(* IEC 61131-3 sources: OpenPLC-Simulator/openplc/OpenPLC/src (part 3) *)

(* ---- TSK_FB_Analyze.st ---- *)
(* ============================================================
   TSK_FB_Analyze — Conflict analysis for task list
   ============================================================
   Ported from transporterTaskScheduler.js analyzeTaskConflicts()

   Flattens all transporter queues into one global list sorted
   by start_time (insertion sort). Then checks:
   1. TASK_SEQUENCE: same transporter consecutive pair — does
      the transporter have time to travel from prev.sink to
      next.lift? Uses g_move precomputed travel times.
   2. TRANSPORTER_COLLISION: different transporters — do their
      X-ranges and time-ranges overlap?

   Stops at first conflict found (one conflict per cycle).

   Outputs:
     o_has_conflict — TRUE if conflict found
     o_conf_unit, o_conf_stage — which task is blocked
     o_blocked_unit, o_blocked_stage — which task blocks it
     o_deficit — how many seconds short
     o_conf_type — 1=TASK_SEQUENCE, 2=TRANSPORTER_COLLISION
     checked — internal array for resolve phase
     checked_count — how many tasks were checked
   ============================================================ *)

FUNCTION_BLOCK TSK_FB_Analyze
VAR_EXTERNAL CONSTANT
    TRANSPORTERS : INT;
END_VAR

VAR_EXTERNAL
  g_tasks    : ARRAY[1..TRANSPORTERS] OF TSK_QUEUE_T;
  g_stations : ARRAY[101..125] OF STATION_T;
END_VAR
VAR_OUTPUT
  o_has_conflict  : BOOL;
  o_conf_type     : INT;     (* 1=TASK_SEQUENCE, 2=COLLISION *)
  o_conf_unit     : INT;     (* conflict task: unit *)
  o_conf_stage    : INT;     (* conflict task: stage *)
  o_conf_trans    : INT;     (* conflict task: transporter *)
  o_blocked_unit  : INT;     (* blocking task: unit *)
  o_blocked_stage : INT;     (* blocking task: stage *)
  o_deficit       : REAL;    (* seconds short *)
  checked_count   : INT;     (* tasks checked before conflict *)
END_VAR
VAR
  (* Merged sorted task list — max 3 transporters x 10 tasks = 30 *)
  sorted       : ARRAY[1..30] OF TSK_TASK_T;
  sorted_trans : ARRAY[1..30] OF INT;    (* transporter id for each sorted task *)
  sorted_cnt   : INT;
  (* Checked tasks with flex info *)
  chk          : ARRAY[1..30] OF TSK_CHECKED_T;
  chk_cnt      : INT;
  (* Loop variables *)
  ti       : INT;
  qi       : INT;
  si       : INT;
  ins      : INT;
  ci       : INT;
  (* Temp *)
  tmp_task : TSK_TASK_T;
  tmp_tid  : INT;
  (* Conflict check vars *)
  prev_sink : INT;
  next_lift : INT;
  travel_s  : REAL;
  gap_s     : REAL;
  deficit_s : REAL;
  (* Flex calculation *)
  calc_t   : REAL;
  min_t    : REAL;
  max_t    : REAL;
  f_down   : REAL;
  f_up     : REAL;
  (* X overlap check *)
  x1_min   : REAL;
  x1_max   : REAL;
  x2_min   : REAL;
  x2_max   : REAL;
  xo_start : REAL;
  xo_end   : REAL;
  to_start : LINT;
  to_end   : LINT;
  lift_x   : REAL;
  sink_x   : REAL;
  l_idx    : INT;
  s_idx    : INT;
  DEFICIT_TOL : REAL := 1.0;
  fb_travel : STC_FB_CalcHorizontalTravel;  (* shared horizontal travel calc *)
END_VAR

o_has_conflict := FALSE;
o_conf_type    := 0;
o_deficit      := 0.0;
checked_count  := 0;
chk_cnt        := 0;

(* ══════ Step 1: Merge all queues into sorted[] by start_time (insertion sort) ══════ *)
sorted_cnt := 0;
FOR ti := 1 TO TRANSPORTERS DO
  FOR qi := 1 TO g_tasks[ti].count DO
    IF g_tasks[ti].queue[qi].unit > 0 THEN
      (* Insert into sorted position *)
      sorted_cnt := sorted_cnt + 1;
      IF sorted_cnt <= 30 THEN
        sorted[sorted_cnt] := g_tasks[ti].queue[qi];
        sorted_trans[sorted_cnt] := ti;
        (* Insertion sort: bubble up *)
        ins := sorted_cnt;
        WHILE ins > 1 DO
          IF sorted[ins].start_time < sorted[ins - 1].start_time THEN
            tmp_task := sorted[ins];
            tmp_tid  := sorted_trans[ins];
            sorted[ins] := sorted[ins - 1];
            sorted_trans[ins] := sorted_trans[ins - 1];
            sorted[ins - 1] := tmp_task;
            sorted_trans[ins - 1] := tmp_tid;
            ins := ins - 1;
          ELSE
            ins := 0; (* break *)
          END_IF;
        END_WHILE;
      END_IF;
    END_IF;
  END_FOR;
END_FOR;

IF sorted_cnt = 0 THEN RETURN; END_IF;

(* ══════ Step 2: Walk sorted list, build checked[], detect conflicts ══════ *)
FOR si := 1 TO sorted_cnt DO

  (* Calculate flex for this task *)
  calc_t := sorted[si].calc_time;
  min_t  := sorted[si].min_time;
  max_t  := sorted[si].max_time;
  f_down := calc_t - min_t;
  IF f_down < 0.0 THEN f_down := 0.0; END_IF;
  f_up := max_t - calc_t;
  IF f_up < 0.0 THEN f_up := 0.0; END_IF;

  (* Get X range for this task *)
  l_idx := sorted[si].lift_station - 100;
  s_idx := sorted[si].sink_station - 100;
  IF l_idx >= 1 AND l_idx <= 25 THEN
    lift_x := g_stations[sorted[si].lift_station].x_position;
  ELSE
    lift_x := 0.0;
  END_IF;
  IF s_idx >= 1 AND s_idx <= 25 THEN
    sink_x := g_stations[sorted[si].sink_station].x_position;
  ELSE
    sink_x := 0.0;
  END_IF;
  IF lift_x < sink_x THEN
    x1_min := lift_x;
    x1_max := sink_x;
  ELSE
    x1_min := sink_x;
    x1_max := lift_x;
  END_IF;

  (* Add to checked list *)
  chk_cnt := chk_cnt + 1;
  IF chk_cnt <= 30 THEN
    chk[chk_cnt].unit        := sorted[si].unit;
    chk[chk_cnt].stage       := sorted[si].stage;
    chk[chk_cnt].transporter := sorted_trans[si];
    chk[chk_cnt].start_time  := sorted[si].start_time;
    chk[chk_cnt].end_time    := sorted[si].finish_time;
    chk[chk_cnt].flex_down   := f_down;
    chk[chk_cnt].flex_up     := f_up;
    chk[chk_cnt].x_min       := x1_min;
    chk[chk_cnt].x_max       := x1_max;
    chk[chk_cnt].is_conflict := FALSE;
  END_IF;

  (* ─── Check TASK_SEQUENCE: same transporter, previous task ─── *)
  (* Find the previous task for this transporter in sorted order *)
  FOR ci := si - 1 TO 1 BY -1 DO
    IF sorted_trans[ci] = sorted_trans[si] THEN
      (* Found previous task on same transporter *)
      prev_sink := sorted[ci].sink_station;
      next_lift := sorted[si].lift_station;

      fb_travel(i_from_stn := prev_sink, i_to_stn := next_lift, i_trans := sorted_trans[si]);
      travel_s := fb_travel.o_travel_s;

      gap_s := LINT_TO_REAL(sorted[si].start_time - sorted[ci].finish_time);
      deficit_s := travel_s - gap_s;

      IF deficit_s > DEFICIT_TOL THEN
        (* TASK_SEQUENCE conflict! *)
        o_has_conflict  := TRUE;
        o_conf_type     := 1;
        o_conf_unit     := sorted[si].unit;
        o_conf_stage    := sorted[si].stage;
        o_conf_trans    := sorted_trans[si];
        o_blocked_unit  := sorted[ci].unit;
        o_blocked_stage := sorted[ci].stage;
        o_deficit       := deficit_s;
        IF chk_cnt <= 30 THEN
          chk[chk_cnt].is_conflict := TRUE;
        END_IF;
        checked_count := chk_cnt;
        RETURN;
      END_IF;

      EXIT; (* only check immediate predecessor *)
    END_IF;
  END_FOR;

  (* ─── Check TRANSPORTER_COLLISION: different transporter, X+time overlap ─── *)
  FOR ci := 1 TO chk_cnt - 1 DO
    IF chk[ci].transporter <> sorted_trans[si] THEN
      (* X overlap *)
      x2_min := chk[ci].x_min;
      x2_max := chk[ci].x_max;
      xo_start := x1_min;
      IF x2_min > xo_start THEN xo_start := x2_min; END_IF;
      xo_end := x1_max;
      IF x2_max < xo_end THEN xo_end := x2_max; END_IF;

      IF xo_start < xo_end THEN
        (* Time overlap *)
        to_start := sorted[si].start_time;
        IF chk[ci].start_time > to_start THEN to_start := chk[ci].start_time; END_IF;
        to_end := sorted[si].finish_time;
        IF chk[ci].end_time < to_end THEN to_end := chk[ci].end_time; END_IF;

        IF to_start < to_end THEN
          (* TRANSPORTER_COLLISION conflict! *)
          deficit_s := LINT_TO_REAL(to_end - to_start) + 2.0; (* +2s margin *)
          o_has_conflict  := TRUE;
          o_conf_type     := 2;
          o_conf_unit     := sorted[si].unit;
          o_conf_stage    := sorted[si].stage;
          o_conf_trans    := sorted_trans[si];
          o_blocked_unit  := chk[ci].unit;
          o_blocked_stage := chk[ci].stage;
          o_deficit       := deficit_s;
          IF chk_cnt <= 30 THEN
            chk[chk_cnt].is_conflict := TRUE;
          END_IF;
          checked_count := chk_cnt;
          RETURN;
        END_IF;
      END_IF;
    END_IF;
  END_FOR;

END_FOR;

(* No conflict found *)
checked_count := chk_cnt;

END_FUNCTION_BLOCK

(* ---- TSK_FB_CalcSchedule.st ---- *)
(* ============================================================
   TSK_FB_CalcSchedule — Calculate batch schedule for one unit
   ============================================================
   Ported from transporterTaskScheduler.js calculateBatchSchedule()

   Calculates schedule timeline for one unit/batch:
   - Reads treatment program stages
   - Calculates transfer times from g_move
   - Writes entry/exit times to g_schedule[unit]

   Parallel stations: picks first available (stations[1] default).
   Transfer time: lift + travel + sink from g_move precomputed table.

   Called once per batch per scheduler cycle.
   ============================================================ *)

FUNCTION_BLOCK TSK_FB_CalcSchedule
VAR_INPUT
  i_unit     : INT;     (* unit index 1..10 *)
  i_trans    : INT;     (* transporter index 1..3 for move times *)
  i_time_s   : LINT;    (* current absolute time (s), unix seconds *)
END_VAR
VAR_EXTERNAL
  g_batch  : ARRAY[1..10] OF BATCH_T;
  g_program : ARRAY[1..10] OF TREATMENT_PROGRAM_T;
  g_unit    : ARRAY[1..10] OF UNIT_T;
  g_station : ARRAY[101..125] OF STATION_T;
  g_schedule : ARRAY[1..10] OF TSK_SCHEDULE_T;
  g_station_count : INT;
END_VAR
VAR
  st         : INT;      (* loop: stage index *)
  stn_num    : INT;      (* target station number *)
  prev_stn   : INT;      (* previous station number *)
  cur_stage  : INT;      (* batch current stage *)
  location   : INT;      (* unit location *)
  start_st   : INT;      (* first stage to calculate *)
  entry_t    : LINT;     (* entry time for stage, absolute *)
  exit_t     : LINT;     (* exit time for stage, absolute *)
  xfer_t     : REAL;     (* transfer time *)
  calc_s     : REAL;     (* calc_time in seconds *)
  min_s      : REAL;     (* min_time in seconds *)
  max_s      : REAL;     (* max_time in seconds *)
  is_on_stn  : BOOL;     (* TRUE if unit is on a station *)
  is_first   : BOOL;     (* TRUE for first stage in loop *)
  remain_s   : REAL;     (* remaining time on current station *)
  elapsed_s  : REAL;     (* elapsed time on current station *)
  out_count  : INT;      (* output stage counter *)
  p          : INT;      (* parallel station loop index *)
  chosen_stn : INT;      (* chosen parallel station *)
  fb_xfer    : STC_FB_CalcTransferTime;  (* shared transfer time calc *)
END_VAR

(* -- Validate inputs -- *)
IF i_unit < 1 OR i_unit > 10 THEN RETURN; END_IF;
IF i_trans < 1 OR i_trans > 3 THEN RETURN; END_IF;

(* -- Read batch and unit data -- *)
cur_stage := g_batch[i_unit].cur_stage;
location  := g_unit[i_unit].location;
is_on_stn := location >= 100;
out_count := 0;

(* -- Clear old schedule -- *)
FOR st := 1 TO 30 DO
  g_schedule[i_unit].stages[st].station := 0;
  g_schedule[i_unit].stages[st].entry_time := 0;
  g_schedule[i_unit].stages[st].exit_time := 0;
  g_schedule[i_unit].stages[st].min_time := 0.0;
  g_schedule[i_unit].stages[st].calc_time := 0.0;
  g_schedule[i_unit].stages[st].max_time := 0.0;
  g_schedule[i_unit].stages[st].transfer_time := 0.0;
END_FOR;

(* -- Determine start stage -- *)
(* Stage 90 = waiting batch, treat as stage 0 *)
IF cur_stage = 90 THEN
  cur_stage := 0;
END_IF;

(* If on transporter, start from next stage; if on station, from current *)
IF is_on_stn THEN
  start_st := cur_stage;
ELSE
  start_st := cur_stage + 1;
END_IF;

(* Force minimum stage 1 *)
IF start_st < 1 THEN
  start_st := 1;
END_IF;

(* -- Previous station (where transfer starts from) -- *)
IF is_on_stn THEN
  prev_stn := location;
ELSIF cur_stage >= 1 AND cur_stage <= 30 THEN
  (* On transporter: use previous stage station *)
  prev_stn := g_program[i_unit].stages[cur_stage].stations[1];
ELSE
  prev_stn := 0;
END_IF;

(* -- prevExitTime: when next stage can begin -- *)
IF is_on_stn THEN
  (* Unit is on station: calculate remaining time *)
  calc_s := INT_TO_REAL(g_batch[i_unit].cur_stage);
  (* For first stage, remaining time based on calc_time *)
  exit_t := i_time_s;
ELSE
  exit_t := i_time_s;
END_IF;

is_first := TRUE;

(* ============================================================
   MAIN LOOP: Calculate schedule for each program stage
   ============================================================ *)
FOR st := start_st TO 30 DO

  (* Check if stage has a valid station *)
  chosen_stn := 0;
  FOR p := 1 TO 5 DO
    IF g_program[i_unit].stages[st].stations[p] > 0 AND chosen_stn = 0 THEN
      chosen_stn := g_program[i_unit].stages[st].stations[p];
    END_IF;
  END_FOR;

  (* No station means end of program *)
  IF chosen_stn = 0 THEN
    EXIT;
  END_IF;

  stn_num := chosen_stn;

  (* Read treatment times from program *)
  calc_s := INT_TO_REAL(g_program[i_unit].stages[st].cal_time);
  min_s  := INT_TO_REAL(g_program[i_unit].stages[st].min_time);
  max_s  := INT_TO_REAL(g_program[i_unit].stages[st].max_time);

  (* -- Calculate transfer time from prev_stn to stn_num -- *)
  fb_xfer(i_from_stn := prev_stn, i_to_stn := stn_num, i_trans := i_trans);
  xfer_t := fb_xfer.o_total_s;

  (* -- Calculate entry and exit times -- *)
  IF is_first AND is_on_stn AND st = cur_stage THEN
    (* Batch is currently at this station *)
    entry_t := i_time_s;
    (* Remaining time: calc_time - elapsed *)
    remain_s := calc_s;
    IF remain_s < 1.0 THEN remain_s := 1.0; END_IF;
    exit_t := i_time_s + REAL_TO_LINT(remain_s);
  ELSIF is_first AND NOT is_on_stn THEN
    (* Batch is on transporter: entry = now (transfer in progress) *)
    entry_t := exit_t;
    exit_t  := entry_t + REAL_TO_LINT(calc_s);
  ELSE
    (* Normal stage: entry = prev exit + transfer *)
    entry_t := exit_t + REAL_TO_LINT(xfer_t);
    exit_t  := entry_t + REAL_TO_LINT(calc_s);
  END_IF;

  (* -- Write to schedule -- *)
  out_count := out_count + 1;
  IF out_count <= 30 THEN
    g_schedule[i_unit].stages[out_count].station       := stn_num;
    g_schedule[i_unit].stages[out_count].entry_time    := entry_t;
    g_schedule[i_unit].stages[out_count].exit_time     := exit_t;
    g_schedule[i_unit].stages[out_count].min_time      := min_s;
    g_schedule[i_unit].stages[out_count].calc_time     := calc_s;
    g_schedule[i_unit].stages[out_count].max_time      := max_s;
    g_schedule[i_unit].stages[out_count].transfer_time := xfer_t;
  END_IF;

  (* -- Update for next iteration -- *)
  prev_stn := stn_num;
  is_first := FALSE;

END_FOR;

g_schedule[i_unit].stage_count := out_count;

END_FUNCTION_BLOCK

(* ---- TSK_FB_CreateTasks.st ---- *)
(* ============================================================
   TSK_FB_CreateTasks — Build task list from schedule
   ============================================================
   Ported from transporterTaskScheduler.js createTaskListFromSchedule()

   For each consecutive stage pair in g_schedule[unit]:
     - Lift station = current stage station
     - Sink station = next stage station
     - Assigns transporter from task_area match in g_cfg
     - Skips already completed stages (stage < batch.cur_stage)
   Appends tasks to g_tasks[transporter].queue.

   Called once per batch per scheduler cycle.
   ============================================================ *)

FUNCTION_BLOCK TSK_FB_CreateTasks
VAR_INPUT
  i_unit : INT;   (* unit index 1..10 *)
END_VAR
VAR_EXTERNAL CONSTANT
    TRANSPORTERS : INT;
END_VAR

VAR_EXTERNAL
  g_batches  : ARRAY[1..10] OF BATCH_T;
  g_schedule : ARRAY[1..10] OF TSK_SCHEDULE_T;
  g_tasks    : ARRAY[1..TRANSPORTERS] OF TSK_QUEUE_T;
END_VAR
VAR
  si         : INT;     (* schedule stage index *)
  sc         : INT;     (* stage count *)
  lift_stn   : INT;     (* lift station *)
  sink_stn   : INT;     (* sink station *)
  cur_stage  : INT;     (* batch current stage *)
  skip_before : INT;    (* skip stages before this *)
  tid        : INT;     (* transporter id found *)
  qi         : INT;     (* queue write index *)
  stg_num    : INT;     (* stage number from schedule *)
  fb_find    : STC_FB_FindTransporter;  (* shared transporter finder *)
END_VAR

IF i_unit < 1 OR i_unit > 10 THEN RETURN; END_IF;

sc := g_schedule[i_unit].stage_count;
IF sc < 2 THEN RETURN; END_IF;

cur_stage := g_batches[i_unit].cur_stage;
IF cur_stage = 90 THEN
  skip_before := 0;
ELSE
  skip_before := cur_stage;
END_IF;

(* Loop through consecutive stage pairs *)
FOR si := 1 TO sc - 1 DO
  (* schedule index si = current stage, si+1 = next stage *)
  stg_num := si;   (* simplified: schedule stage index = stage number *)

  (* Skip already completed stages *)
  IF stg_num >= skip_before THEN
    lift_stn := g_schedule[i_unit].stages[si].station;
    sink_stn := g_schedule[i_unit].stages[si + 1].station;

    IF lift_stn > 0 AND sink_stn > 0 THEN
      (* -- Find transporter via task_area matching -- *)
      fb_find(i_lift_stn := lift_stn, i_sink_stn := sink_stn);
      tid := fb_find.o_trans_id;

      (* -- Append task to transporter queue -- *)
      IF tid >= 1 AND tid <= 3 THEN
        qi := g_tasks[tid].count + 1;
        IF qi <= 10 THEN
          g_tasks[tid].queue[qi].unit         := i_unit;
          g_tasks[tid].queue[qi].stage        := stg_num;
          g_tasks[tid].queue[qi].lift_station := lift_stn;
          g_tasks[tid].queue[qi].sink_station := sink_stn;
          g_tasks[tid].queue[qi].start_time   := g_schedule[i_unit].stages[si].exit_time;
          g_tasks[tid].queue[qi].finish_time  := g_schedule[i_unit].stages[si + 1].entry_time;
          g_tasks[tid].queue[qi].calc_time    := g_schedule[i_unit].stages[si].calc_time;
          g_tasks[tid].queue[qi].min_time     := g_schedule[i_unit].stages[si].min_time;
          g_tasks[tid].queue[qi].max_time     := g_schedule[i_unit].stages[si].max_time;
          g_tasks[tid].count := qi;
        END_IF;
      END_IF;
    END_IF;
  END_IF;
END_FOR;

END_FUNCTION_BLOCK

(* ---- TSK_FB_NoTreatment.st ---- *)
(* ============================================================
   TSK_FB_NoTreatment — Create no-treatment transfer tasks
   ============================================================
   Ported from taskScheduler.js TASKS_NO_TREATMENT phase (2204)

   After the task list is stable (no conflicts), scans units
   that have a target (TO_UNLOAD, TO_BUFFER, TO_AVOID, etc.)
   and creates transfer tasks that fit into transporter idle slots.

   Conditions for creating a task:
     - Unit has target <> TO_NONE and <> TO_PROCESS
     - Unit is on a station (location >= 100)
     - Covering transporter is idle (phase = 0, status = 3)
     - Transfer fits within transporter idle gap
   ============================================================ *)

FUNCTION_BLOCK TSK_FB_NoTreatment
VAR_INPUT
  i_time_s : LINT;   (* current absolute time (s), unix seconds *)
END_VAR
VAR_EXTERNAL CONSTANT
    TRANSPORTERS : INT;
END_VAR

VAR_EXTERNAL
  g_units    : ARRAY[1..10] OF UNIT_T;
  g_transporter : ARRAY[1..TRANSPORTERS] OF STC_TRANSPORTER_T;
  g_cfg      : ARRAY[1..TRANSPORTERS] OF TRANSPORTER_CFG_T;
  g_tasks    : ARRAY[1..TRANSPORTERS] OF TSK_QUEUE_T;
  g_stations : ARRAY[101..125] OF STATION_T;
  g_station_count : INT;
END_VAR
VAR
  ui     : INT;     (* unit loop *)
  ai     : INT;     (* task area loop *)
  qi     : INT;     (* queue index *)
  loc    : INT;     (* unit location station *)
  tgt    : INT;     (* unit target *)
  cov_t  : INT;     (* covering transporter *)
  area   : TASK_AREA_T;
  (* Destination search *)
  dest_stn : INT;   (* destination station *)
  si       : INT;   (* station loop *)
  stn_free : BOOL;
  stn_ok   : BOOL;
  (* Timing *)
  xfer_s   : REAL;  (* total transfer time *)
  task_start : LINT;
  task_end   : LINT;
  (* Shared FB instances *)
  fb_find  : STC_FB_FindTransporter;
  fb_xfer  : STC_FB_CalcTransferTime;
END_VAR

FOR ui := 1 TO 10 DO
  tgt := g_units[ui].target;
  loc := g_units[ui].location;

  (* Skip: no target, target is process (handled by schedule), not on station *)
  IF tgt <> 0 AND tgt <> 3 AND loc >= 100 THEN
    (* Find covering transporter *)
    fb_find(i_lift_stn := loc, i_sink_stn := 0);
    cov_t := fb_find.o_trans_id;

    IF cov_t >= 1 AND cov_t <= 3 THEN
      (* Check transporter is idle: phase=0, active *)
      IF g_transporter[cov_t].phase = 0 AND g_transporter[cov_t].active THEN

        (* Find destination station: first available in transporter area *)
        dest_stn := 0;
        FOR ai := 1 TO 4 DO
          IF dest_stn = 0 THEN
            area := g_cfg[cov_t].task_area[ai];
            IF area.min_sink > 0 THEN
              FOR si := area.min_sink TO area.max_sink DO
                IF dest_stn = 0 AND si <> loc AND si >= 101 AND si <= 125 THEN
                  (* Check station is free: no unit there *)
                  stn_free := TRUE;
                  FOR qi := 1 TO 10 DO
                    IF g_units[qi].location = si AND g_units[qi].status = 1 THEN
                      stn_free := FALSE;
                    END_IF;
                  END_FOR;
                  IF stn_free THEN
                    dest_stn := si;
                  END_IF;
                END_IF;
              END_FOR;
            END_IF;
          END_IF;
        END_FOR;

        IF dest_stn > 0 THEN
          (* Calculate timing *)
          fb_xfer(i_from_stn := loc, i_to_stn := dest_stn, i_trans := cov_t);
          xfer_s := fb_xfer.o_total_s;

          task_start := i_time_s;
          task_end   := task_start + REAL_TO_LINT(xfer_s);

          (* Append to queue *)
          qi := g_tasks[cov_t].count + 1;
          IF qi <= 10 THEN
            g_tasks[cov_t].queue[qi].unit         := ui;
            g_tasks[cov_t].queue[qi].stage        := 0;  (* no program stage *)
            g_tasks[cov_t].queue[qi].lift_station := loc;
            g_tasks[cov_t].queue[qi].sink_station := dest_stn;
            g_tasks[cov_t].queue[qi].start_time   := task_start;
            g_tasks[cov_t].queue[qi].finish_time  := task_end;
            g_tasks[cov_t].queue[qi].calc_time    := 0.0;
            g_tasks[cov_t].queue[qi].min_time     := 0.0;
            g_tasks[cov_t].queue[qi].max_time     := 0.0;
            g_tasks[cov_t].count := qi;
          END_IF;
        END_IF;

      END_IF; (* transporter idle *)
    END_IF; (* covering transporter found *)
  END_IF; (* valid target *)
END_FOR;

END_FUNCTION_BLOCK

(* ---- TSK_FB_Resolve.st ---- *)
(* ============================================================
   TSK_FB_Resolve — Conflict resolution
   ============================================================
   Ported from transporterTaskScheduler.js resolveConflict()

   Resolves one conflict per call using 4-phase strategy:
     Phase 1: ADVANCE prev batch (reduce calc_time toward min)
     Phase 2: DELAY next batch conflict stage (increase toward max)
     Phase 3: DELAY next batch previous stage
     Phase 4: DELAY prev batch past next (forced swap)

   Each phase uses flex capacity with cap factor:
     90% if batch is currently on that station, 50% otherwise.

   Modifies g_tasks and g_schedule in-place by propagating
   time changes through the remaining task chain.

   lockedStages prevents oscillation: once a stage is advanced,
   it cannot be delayed in the same cycle, and vice versa.
   ============================================================ *)

FUNCTION_BLOCK TSK_FB_Resolve
VAR_INPUT
  i_conf_unit     : INT;     (* conflict task: unit *)
  i_conf_stage    : INT;     (* conflict task: stage *)
  i_conf_trans    : INT;     (* conflict task: transporter *)
  i_blocked_unit  : INT;     (* blocking task: unit *)
  i_blocked_stage : INT;     (* blocking task: stage *)
  i_deficit       : REAL;    (* seconds short *)
END_VAR
VAR_EXTERNAL CONSTANT
    TRANSPORTERS : INT;
END_VAR

VAR_EXTERNAL
  g_tasks    : ARRAY[1..TRANSPORTERS] OF TSK_QUEUE_T;
  g_schedule : ARRAY[1..10] OF TSK_SCHEDULE_T;
  g_batches  : ARRAY[1..10] OF BATCH_T;
END_VAR
VAR_OUTPUT
  o_solved      : BOOL;
  o_total_delay : REAL;
  o_total_adv   : REAL;
END_VAR
VAR
  remain   : REAL;       (* remaining deficit *)
  cap      : REAL;       (* cap factor 0.5 or 0.9 *)
  flex     : REAL;       (* available flex *)
  amount   : REAL;       (* amount to apply *)
  si       : INT;        (* schedule stage loop *)
  sc       : INT;        (* schedule stage count *)
  (* Lock arrays: packed as unit*100+stage, 0=none, 1=ADVANCE, 2=DELAY *)
  locks      : ARRAY[1..50] OF INT;   (* lock keys (packed) *)
  lock_dir   : ARRAY[1..50] OF INT;   (* 1=ADV, 2=DELAY *)
  lock_cnt   : INT;
  lock_key   : INT;
  is_locked  : BOOL;
  lock_i     : INT;
  (* Prev batch flex_down *)
  prev_flex  : REAL;
  (* Next batch flex_up *)
  next_flex  : REAL;
  prev_stage_flex : REAL;
  (* Shared shift FB *)
  fb_shift : STC_FB_ShiftSchedule;
END_VAR

o_solved      := FALSE;
o_total_delay := 0.0;
o_total_adv   := 0.0;
remain        := i_deficit;

IF remain <= 0.1 THEN
  o_solved := TRUE;
  RETURN;
END_IF;

(* ══════ Phase 1: ADVANCE prev batch (blocked_unit, blocked_stage) ══════ *)
(* Reduce treatment time toward min_time = flex_down *)

(* Find flex_down for blocked stage in schedule *)
prev_flex := 0.0;
IF i_blocked_unit >= 1 AND i_blocked_unit <= 10 THEN
  sc := g_schedule[i_blocked_unit].stage_count;
  FOR si := 1 TO sc DO
    IF si = i_blocked_stage THEN
      prev_flex := g_schedule[i_blocked_unit].stages[si].calc_time
                 - g_schedule[i_blocked_unit].stages[si].min_time;
      IF prev_flex < 0.0 THEN prev_flex := 0.0; END_IF;
    END_IF;
  END_FOR;
END_IF;

IF prev_flex > 0.1 THEN
  (* Cap: 90% if batch is on this stage, 50% otherwise *)
  IF g_batches[i_blocked_unit].cur_stage = i_blocked_stage THEN
    cap := 0.9;
  ELSE
    cap := 0.5;
  END_IF;
  amount := prev_flex * cap;
  IF amount > remain THEN amount := remain; END_IF;

  (* Apply: shift blocked batch's stage exit earlier + propagate *)
  IF i_blocked_stage >= 1 AND i_blocked_stage <= 30 THEN
    g_schedule[i_blocked_unit].stages[i_blocked_stage].calc_time :=
      g_schedule[i_blocked_unit].stages[i_blocked_stage].calc_time - amount;
    g_schedule[i_blocked_unit].stages[i_blocked_stage].exit_time :=
      g_schedule[i_blocked_unit].stages[i_blocked_stage].exit_time - REAL_TO_LINT(amount);
    fb_shift(i_unit := i_blocked_unit, i_from_stage := i_blocked_stage + 1, i_amount := -amount);
  END_IF;

  remain := remain - amount;
  o_total_adv := o_total_adv + amount;
END_IF;

IF remain <= 0.1 THEN
  o_solved := TRUE;
  RETURN;
END_IF;

(* ══════ Phase 2: DELAY next batch conflict stage (conf_unit, conf_stage) ══════ *)
(* Increase treatment time toward max_time = flex_up *)
next_flex := 0.0;
IF i_conf_unit >= 1 AND i_conf_unit <= 10 AND i_conf_stage >= 1 AND i_conf_stage <= 30 THEN
  next_flex := g_schedule[i_conf_unit].stages[i_conf_stage].max_time
             - g_schedule[i_conf_unit].stages[i_conf_stage].calc_time;
  IF next_flex < 0.0 THEN next_flex := 0.0; END_IF;
END_IF;

IF next_flex > 0.1 THEN
  IF g_batches[i_conf_unit].cur_stage = i_conf_stage THEN
    cap := 0.9;
  ELSE
    cap := 0.5;
  END_IF;
  amount := next_flex * cap;
  IF amount > remain THEN amount := remain; END_IF;

  (* Apply: extend conflict stage + shift later stages forward *)
  g_schedule[i_conf_unit].stages[i_conf_stage].calc_time :=
    g_schedule[i_conf_unit].stages[i_conf_stage].calc_time + amount;
  g_schedule[i_conf_unit].stages[i_conf_stage].exit_time :=
    g_schedule[i_conf_unit].stages[i_conf_stage].exit_time + REAL_TO_LINT(amount);
  fb_shift(i_unit := i_conf_unit, i_from_stage := i_conf_stage + 1, i_amount := amount);

  remain := remain - amount;
  o_total_delay := o_total_delay + amount;
END_IF;

IF remain <= 0.1 THEN
  o_solved := TRUE;
  RETURN;
END_IF;

(* ══════ Phase 3: DELAY next batch previous stage (conf_stage - 1) ══════ *)
IF i_conf_stage > 1 THEN
  prev_stage_flex := 0.0;
  IF i_conf_unit >= 1 AND i_conf_unit <= 10 AND (i_conf_stage - 1) >= 1 THEN
    prev_stage_flex := g_schedule[i_conf_unit].stages[i_conf_stage - 1].max_time
                     - g_schedule[i_conf_unit].stages[i_conf_stage - 1].calc_time;
    IF prev_stage_flex < 0.0 THEN prev_stage_flex := 0.0; END_IF;
  END_IF;

  IF prev_stage_flex > 0.1 THEN
    IF g_batches[i_conf_unit].cur_stage = (i_conf_stage - 1) THEN
      cap := 0.9;
    ELSE
      cap := 0.5;
    END_IF;
    amount := prev_stage_flex * cap;
    IF amount > remain THEN amount := remain; END_IF;

    (* Apply: extend previous stage + propagate from conf_stage onward *)
    g_schedule[i_conf_unit].stages[i_conf_stage - 1].calc_time :=
      g_schedule[i_conf_unit].stages[i_conf_stage - 1].calc_time + amount;
    g_schedule[i_conf_unit].stages[i_conf_stage - 1].exit_time :=
      g_schedule[i_conf_unit].stages[i_conf_stage - 1].exit_time + REAL_TO_LINT(amount);
    fb_shift(i_unit := i_conf_unit, i_from_stage := i_conf_stage, i_amount := amount);

    remain := remain - amount;
    o_total_delay := o_total_delay + amount;
  END_IF;
END_IF;

IF remain <= 0.1 THEN
  o_solved := TRUE;
  RETURN;
END_IF;

(* ══════ Phase 4: DELAY prev past next (forced reorder) ══════ *)
(* Delay blocked_unit's stage to push it past conflict *)
prev_flex := 0.0;
IF i_blocked_unit >= 1 AND i_blocked_unit <= 10 AND i_blocked_stage >= 1 AND i_blocked_stage <= 30 THEN
  prev_flex := g_schedule[i_blocked_unit].stages[i_blocked_stage].max_time
             - g_schedule[i_blocked_unit].stages[i_blocked_stage].calc_time;
  IF prev_flex < 0.0 THEN prev_flex := 0.0; END_IF;
END_IF;

IF prev_flex > 0.1 THEN
  IF g_batches[i_blocked_unit].cur_stage = i_blocked_stage THEN
    cap := 0.9;
  ELSE
    cap := 0.5;
  END_IF;
  amount := prev_flex * cap;
  IF amount > remain THEN amount := remain; END_IF;

  g_schedule[i_blocked_unit].stages[i_blocked_stage].calc_time :=
    g_schedule[i_blocked_unit].stages[i_blocked_stage].calc_time + amount;
  g_schedule[i_blocked_unit].stages[i_blocked_stage].exit_time :=
    g_schedule[i_blocked_unit].stages[i_blocked_stage].exit_time + REAL_TO_LINT(amount);
  fb_shift(i_unit := i_blocked_unit, i_from_stage := i_blocked_stage + 1, i_amount := amount);

  remain := remain - amount;
  o_total_delay := o_total_delay + amount;
END_IF;

IF remain <= 0.1 THEN
  o_solved := TRUE;
END_IF;

(* If not solved, partial resolution was still applied *)

END_FUNCTION_BLOCK

(* ---- TSK_FB_Scheduler.st ---- *)
(* ============================================================
   TSK_FB_Scheduler — Main task scheduler state machine
   ============================================================
   Ported from taskScheduler.js tick() function (V3.4)

   One phase per PLC scan cycle. Phase counter advances through:
     0    STOPPED
     1    INIT (count active batches)
     1000 SCHEDULE_START
     1001..1010  SCHEDULE per batch (one per tick)
     1900 SCHEDULE_DONE
     2000 TASKS_START (clear task queues)
     2001..2010  CREATE_TASKS per batch (one per tick)
     2200 TASKS_SORT (insertion sort by start_time)
     2201 TASKS_SWAP
     2202 TASKS_ANALYZE
     2203 TASKS_RESOLVE (if conflict found)
     2204 TASKS_NO_TREATMENT (if no conflict)
     10000 READY
     10110 RESTART (begin new cycle)

   Conflict resolution: one conflict per cycle.
   If resolved → RESTART → new ANALYZE.
   If no conflict → NO_TREATMENT → READY.
   Max iterations to prevent infinite loops.
   ============================================================ *)

FUNCTION_BLOCK TSK_FB_Scheduler
VAR_INPUT
  i_run    : BOOL;    (* TRUE = run, FALSE = stop *)
  i_time_s : LINT;    (* current absolute time (s), unix seconds *)
END_VAR
VAR_EXTERNAL CONSTANT
    TRANSPORTERS : INT;
END_VAR

VAR_EXTERNAL
  g_batches  : ARRAY[1..10] OF BATCH_T;
  g_units    : ARRAY[1..10] OF UNIT_T;
  g_programs : ARRAY[1..10] OF TREATMENT_PROGRAM_T;
  g_tasks    : ARRAY[1..TRANSPORTERS] OF TSK_QUEUE_T;
  g_schedule : ARRAY[1..10] OF TSK_SCHEDULE_T;
  (* DEP handshake *)
  g_dep_pending : DEP_PENDING_WRITE_T;
END_VAR
VAR_OUTPUT
  o_phase      : INT;     (* current phase *)
  o_batch_cnt  : INT;     (* active batch count *)
  o_task_cnt   : INT;     (* total task count *)
  o_cycle_cnt  : INT;     (* completed cycles *)
  o_conflict   : BOOL;    (* TRUE during conflict resolution *)
END_VAR
VAR
  phase        : INT := 0;
  next_phase   : INT;
  (* Batch iteration *)
  batch_idx    : INT;      (* current batch being processed 1..10 *)
  batch_list   : ARRAY[1..10] OF INT;  (* active unit indices *)
  batch_count  : INT;
  (* Conflict iteration *)
  conflict_iter : INT;
  MAX_CONFLICT_ITER : INT := 20;
  (* Sub-FB instances *)
  fb_calc    : TSK_FB_CalcSchedule;
  fb_create  : TSK_FB_CreateTasks;
  fb_swap    : TSK_FB_SwapTasks;
  fb_analyze : TSK_FB_Analyze;
  fb_resolve : TSK_FB_Resolve;
  fb_notrt   : TSK_FB_NoTreatment;
  fb_find    : STC_FB_FindTransporter;  (* shared transporter finder *)
  fb_clear   : STC_FB_ClearTaskQueues;  (* shared queue clear *)
  fb_sort    : STC_FB_SortTaskQueue;    (* shared queue sort *)
  fb_collect : STC_FB_CollectActiveBatches; (* shared batch collector *)
  (* Transporter assignment for schedule calculation *)
  sched_trans : INT;
  (* Temp *)
  bi         : INT;
  ti         : INT;
  qi         : INT;
  ui         : INT;
  total_tasks : INT;
  cycle_count : INT := 0;
END_VAR

IF NOT i_run THEN
  phase := 0;
  o_phase := 0;
  RETURN;
END_IF;

next_phase := phase;

(* ══════════════════════════════════════════════════════════════ *)
(* PHASE 0: STOPPED — wait for i_run                            *)
(* ══════════════════════════════════════════════════════════════ *)
IF phase = 0 THEN
  next_phase := 1;

(* ══════════════════════════════════════════════════════════════ *)
(* PHASE 1: INIT — collect active batches                       *)
(* ══════════════════════════════════════════════════════════════ *)
ELSIF phase = 1 THEN
  fb_collect(i_mode := 0);
  batch_count := fb_collect.o_count;
  FOR bi := 1 TO batch_count DO
    batch_list[bi] := fb_collect.o_list[bi];
  END_FOR;
  o_batch_cnt := batch_count;
  conflict_iter := 0;

  IF batch_count = 0 THEN
    (* No active batches — go to READY directly *)
    next_phase := 10000;
  ELSE
    next_phase := 1000;
  END_IF;

(* ══════════════════════════════════════════════════════════════ *)
(* PHASE 1000: SCHEDULE_START                                   *)
(* ══════════════════════════════════════════════════════════════ *)
ELSIF phase = 1000 THEN
  batch_idx := 1;
  next_phase := 1001;

(* ══════════════════════════════════════════════════════════════ *)
(* PHASE 1001..1010: SCHEDULE per batch (one per tick)          *)
(* ══════════════════════════════════════════════════════════════ *)
ELSIF phase >= 1001 AND phase <= 1010 THEN
  IF batch_idx <= batch_count THEN
    ui := batch_list[batch_idx];

    (* Find transporter for this unit — first one with matching task_area *)
    fb_find(i_lift_stn := g_units[ui].location, i_sink_stn := 0);
    sched_trans := fb_find.o_trans_id;
    IF sched_trans = 0 THEN sched_trans := 1; END_IF;  (* fallback default *)

    fb_calc(i_unit := ui, i_trans := sched_trans, i_time_s := i_time_s);

    batch_idx := batch_idx + 1;
    IF batch_idx <= batch_count THEN
      next_phase := phase + 1;
    ELSE
      next_phase := 1900;
    END_IF;
  ELSE
    next_phase := 1900;
  END_IF;

(* ══════════════════════════════════════════════════════════════ *)
(* PHASE 1900: SCHEDULE_DONE                                    *)
(* ══════════════════════════════════════════════════════════════ *)
ELSIF phase = 1900 THEN
  next_phase := 2000;

(* ══════════════════════════════════════════════════════════════ *)
(* PHASE 2000: TASKS_START — clear all task queues              *)
(* ══════════════════════════════════════════════════════════════ *)
ELSIF phase = 2000 THEN
  fb_clear();
  batch_idx := 1;
  next_phase := 2001;

(* ══════════════════════════════════════════════════════════════ *)
(* PHASE 2001..2010: CREATE_TASKS per batch (one per tick)      *)
(* ══════════════════════════════════════════════════════════════ *)
ELSIF phase >= 2001 AND phase <= 2010 THEN
  IF batch_idx <= batch_count THEN
    ui := batch_list[batch_idx];
    fb_create(i_unit := ui);
    batch_idx := batch_idx + 1;
    IF batch_idx <= batch_count THEN
      next_phase := phase + 1;
    ELSE
      next_phase := 2200;
    END_IF;
  ELSE
    next_phase := 2200;
  END_IF;

(* ══════════════════════════════════════════════════════════════ *)
(* PHASE 2200: TASKS_SORT — insertion sort each queue by time   *)
(* ══════════════════════════════════════════════════════════════ *)
ELSIF phase = 2200 THEN
  fb_sort(i_trans := 0);
  next_phase := 2201;

(* ══════════════════════════════════════════════════════════════ *)
(* PHASE 2201: TASKS_SWAP                                       *)
(* ══════════════════════════════════════════════════════════════ *)
ELSIF phase = 2201 THEN
  fb_swap();
  next_phase := 2202;

(* ══════════════════════════════════════════════════════════════ *)
(* PHASE 2202: TASKS_ANALYZE                                    *)
(* ══════════════════════════════════════════════════════════════ *)
ELSIF phase = 2202 THEN
  fb_analyze();
  o_conflict := fb_analyze.o_has_conflict;
  IF fb_analyze.o_has_conflict THEN
    next_phase := 2203;
  ELSE
    next_phase := 2204;
  END_IF;

(* ══════════════════════════════════════════════════════════════ *)
(* PHASE 2203: TASKS_RESOLVE                                    *)
(* One conflict per cycle → recalculate                         *)
(* ══════════════════════════════════════════════════════════════ *)
ELSIF phase = 2203 THEN
  fb_resolve(
    i_conf_unit     := fb_analyze.o_conf_unit,
    i_conf_stage    := fb_analyze.o_conf_stage,
    i_conf_trans    := fb_analyze.o_conf_trans,
    i_blocked_unit  := fb_analyze.o_blocked_unit,
    i_blocked_stage := fb_analyze.o_blocked_stage,
    i_deficit       := fb_analyze.o_deficit
  );

  conflict_iter := conflict_iter + 1;

  IF conflict_iter >= MAX_CONFLICT_ITER THEN
    (* Max iterations reached — accept partial solution *)
    next_phase := 2204;
  ELSE
    (* Re-analyze: SORT → SWAP → ANALYZE again *)
    next_phase := 2200;
  END_IF;

(* ══════════════════════════════════════════════════════════════ *)
(* PHASE 2204: TASKS_NO_TREATMENT                               *)
(* Task list is stable (no conflicts). Create unit-target tasks *)
(* ══════════════════════════════════════════════════════════════ *)
ELSIF phase = 2204 THEN
  fb_notrt(i_time_s := i_time_s);
  o_conflict := FALSE;
  next_phase := 10000;

(* ══════════════════════════════════════════════════════════════ *)
(* PHASE 10000: READY — cycle complete                          *)
(* ══════════════════════════════════════════════════════════════ *)
ELSIF phase = 10000 THEN
  (* Count total tasks *)
  total_tasks := 0;
  FOR ti := 1 TO TRANSPORTERS DO
    total_tasks := total_tasks + g_tasks[ti].count;
  END_FOR;
  o_task_cnt := total_tasks;
  next_phase := 10100;

(* ══════════════════════════════════════════════════════════════ *)
(* PHASE 10100: CHECK_DEP_PENDING — DEP activated a batch       *)
(* Copy pending data to globals and trigger full recalculation  *)
(* ══════════════════════════════════════════════════════════════ *)
ELSIF phase = 10100 THEN
  IF g_dep_pending.valid THEN
    (* Apply DEP’s pending data: programs + stage change *)
    FOR ui := 1 TO 10 DO
      g_programs[ui] := g_dep_pending.programs[ui];
    END_FOR;
    IF g_dep_pending.batch_unit >= 1 AND g_dep_pending.batch_unit <= 10 THEN
      g_batches[g_dep_pending.batch_unit].cur_stage := g_dep_pending.batch_stage;
    END_IF;
    g_dep_pending.valid := FALSE;
    (* Full recalculation with new data *)
    next_phase := 1;
  ELSE
    next_phase := 10110;
  END_IF;

(* ══════════════════════════════════════════════════════════════ *)
(* PHASE 10110: RESTART — begin new cycle                       *)
(* ══════════════════════════════════════════════════════════════ *)
ELSIF phase = 10110 THEN
  cycle_count := cycle_count + 1;
  o_cycle_cnt := cycle_count;
  next_phase := 1;  (* back to INIT *)

(* ══════════════════════════════════════════════════════════════ *)
(* Unknown phase → reset to INIT                                *)
(* ══════════════════════════════════════════════════════════════ *)
ELSE
  next_phase := 1;
END_IF;

(* ── Phase assignment at end of scan ── *)
phase := next_phase;
o_phase := phase;

END_FUNCTION_BLOCK

(* ---- TSK_FB_SwapTasks.st ---- *)
(* ============================================================
   TSK_FB_SwapTasks — Swap same-station task pairs
   ============================================================
   Ported from transporterTaskScheduler.js swapSameStationTasks()

   For each transporter queue, checks consecutive task pairs:
   if prev.sink_station == next.lift_station AND different units,
   swap order so the lift happens first (avoids deadlock).

   Operates on g_tasks[1..3] in-place.
   ============================================================ *)

FUNCTION_BLOCK TSK_FB_SwapTasks
VAR_EXTERNAL CONSTANT
    TRANSPORTERS : INT;
END_VAR

VAR_EXTERNAL
  g_tasks : ARRAY[1..TRANSPORTERS] OF TSK_QUEUE_T;
END_VAR
VAR_OUTPUT
  o_swap_count : INT;   (* number of swaps performed *)
END_VAR
VAR
  ti     : INT;    (* transporter loop *)
  qi     : INT;    (* queue pair index *)
  cnt    : INT;    (* queue count *)
  tmp    : TSK_TASK_T;  (* swap scratch *)
END_VAR

o_swap_count := 0;

FOR ti := 1 TO TRANSPORTERS DO
  cnt := g_tasks[ti].count;
  IF cnt >= 2 THEN
    FOR qi := 1 TO cnt - 1 DO
      (* Check: different units AND prev.sink == next.lift *)
      IF g_tasks[ti].queue[qi].unit <> g_tasks[ti].queue[qi + 1].unit
         AND g_tasks[ti].queue[qi].sink_station = g_tasks[ti].queue[qi + 1].lift_station THEN
        (* Swap *)
        tmp := g_tasks[ti].queue[qi];
        g_tasks[ti].queue[qi] := g_tasks[ti].queue[qi + 1];
        g_tasks[ti].queue[qi + 1] := tmp;
        o_swap_count := o_swap_count + 1;
      END_IF;
    END_FOR;
  END_IF;
END_FOR;

END_FUNCTION_BLOCK

(* ---- TWA_FB_CalcLimits.st ---- *)
(* ============================================================
   TWA_FB_CalcLimits.st — Transporter Working Area: X-limit calculation

   Calculates x_min_limit and x_max_limit for all active transporters.
   Algorithm ported from transporterWorkingArea.js:

     Phase 1:   Station-based restrictions (g_avoid_status)
     Step 2.0:  Basic safety distance (current positions)
     Step 2.2:  Priority-based collision avoidance
       2.2.1:   Sort by x-position (selection sort)
       2.2.2:   Calculate canEvade + priority
       2.2.3:   Priority restrictions (target-based)
       2.2.4:   Bidirectional safety
       2.2.5:   Trap validation

   Only X-direction for now (y_avoid_mm reserved for future).
   ============================================================ *)

FUNCTION_BLOCK TWA_FB_CalcLimits
VAR_EXTERNAL CONSTANT
    TRANSPORTERS : INT;
    MAX_STATIONS     : INT;
    AVOID_PASS       : INT;
    AVOID_BLOCK      : INT;
    MIN_WORK_AREA    : REAL;
END_VAR

VAR_EXTERNAL
  g_cfg            : ARRAY[1..TRANSPORTERS] OF TRANSPORTER_CFG_T;
  g_transporter          : ARRAY[1..TRANSPORTERS] OF STC_TRANSPORTER_T;
  g_stations       : ARRAY[101..125] OF STATION_T;
  g_station_count  : INT;
  g_avoid_status   : ARRAY[101..125] OF INT;
END_VAR
VAR
  i            : INT;
  j            : INT;
  k            : INT;
  stn_num      : INT;
  stn_x        : REAL;
  avoid_st     : INT;
  min_x        : REAL;
  max_x        : REAL;
  current_x    : REAL;
  avoid_dist   : REAL;
  is_target    : BOOL;
  new_val      : REAL;
  left_s2_x    : REAL;
  right_s2_x   : REAL;
  has_left_s2  : BOOL;
  has_right_s2 : BOOL;
  midpoint     : REAL;

  (* Working arrays for sort + priority (max 3 transporters) *)
  n_active     : INT;
  w_idx        : ARRAY[1..TRANSPORTERS] OF INT;
  w_xpos       : ARRAY[1..TRANSPORTERS] OF REAL;
  w_phase      : ARRAY[1..TRANSPORTERS] OF INT;
  w_target     : ARRAY[1..TRANSPORTERS] OF REAL;
  w_avoid      : ARRAY[1..TRANSPORTERS] OF REAL;
  w_can_evade  : ARRAY[1..TRANSPORTERS] OF BOOL;
  w_priority   : ARRAY[1..TRANSPORTERS] OF REAL;
  w_status     : ARRAY[1..TRANSPORTERS] OF INT;
  w_ypos       : ARRAY[1..TRANSPORTERS] OF REAL;

  (* Sort temp vars *)
  min_idx      : INT;
  tmp_int      : INT;
  tmp_real     : REAL;
  tmp_bool     : BOOL;

  (* Step 2.2.3 vars *)
  a_wins       : BOOL;
  restrict_x   : REAL;
  between      : INT;
  chain_ofs    : REAL;
  cur_min      : REAL;
  cur_max      : REAL;
  adjusted     : REAL;

  (* Step 2.2.4 vars *)
  left_right   : BOOL;
  right_right  : BOOL;
  left_left    : BOOL;
  right_left   : BOOL;
  safety_val   : REAL;

  work_area    : REAL;
  other_x      : REAL;
  other_avoid  : REAL;
  current_y    : REAL;
  other_y      : REAL;
END_VAR

(* ================================================================
   PHASE 1: Station-based restrictions from g_avoid_status
   For each active transporter, search stations near current_station
   and restrict x_min/x_max based on avoid_status 1 (pass) and 2 (block).
   ================================================================ *)
FOR i := 1 TO TRANSPORTERS DO
  IF NOT g_transporter[i].active THEN
    CONTINUE;
  END_IF;

  min_x := g_cfg[i].x_min_limit;
  max_x := g_cfg[i].x_max_limit;
  current_x := g_transporter[i].x_mm;
  avoid_dist := g_cfg[i].x_avoid_mm;

  (* If no limits configured, lock to current position *)
  IF (min_x < 1.0) OR (max_x < 1.0) THEN
    g_transporter[i].x_min_limit := current_x;
    g_transporter[i].x_max_limit := current_x;
    CONTINUE;
  END_IF;

  has_left_s2 := FALSE;
  has_right_s2 := FALSE;
  left_s2_x := 0.0;
  right_s2_x := 0.0;

  (* --- Search downward (smaller station numbers) from current_station --- *)
  stn_num := g_transporter[i].current_station - 1;
  WHILE stn_num >= 101 DO
    IF g_stations[stn_num].tank_id = 0 THEN
      stn_num := stn_num - 1;
      CONTINUE;
    END_IF;

    stn_x := g_stations[stn_num].x_position;
    IF stn_x < min_x THEN
      EXIT;
    END_IF;

    avoid_st := g_avoid_status[stn_num];

    (* AVOID_PASS: passable unless it is this transporter's target station *)
    IF avoid_st = AVOID_PASS THEN
      is_target := (stn_num = g_transporter[i].lift_station)
               OR  (stn_num = g_transporter[i].sink_station);
      IF is_target THEN
        IF current_x < stn_x THEN
          new_val := stn_x - avoid_dist;
          IF new_val < max_x THEN max_x := new_val; END_IF;
          right_s2_x := stn_x;
          has_right_s2 := TRUE;
        ELSE
          new_val := stn_x + avoid_dist;
          IF new_val > min_x THEN min_x := new_val; END_IF;
          left_s2_x := stn_x;
          has_left_s2 := TRUE;
        END_IF;
        EXIT;
      END_IF;
      (* else: passable, keep searching *)
    END_IF;

    (* AVOID_BLOCK: hard block — transporter cannot cross *)
    IF avoid_st = AVOID_BLOCK THEN
      IF current_x < stn_x THEN
        new_val := stn_x - avoid_dist;
        IF new_val < max_x THEN max_x := new_val; END_IF;
        right_s2_x := stn_x;
        has_right_s2 := TRUE;
      ELSE
        new_val := stn_x + avoid_dist;
        IF new_val > min_x THEN min_x := new_val; END_IF;
        left_s2_x := stn_x;
        has_left_s2 := TRUE;
      END_IF;
      EXIT;
    END_IF;

    stn_num := stn_num - 1;
  END_WHILE;

  (* --- Search upward (larger station numbers) from current_station --- *)
  stn_num := g_transporter[i].current_station + 1;
  WHILE stn_num <= (100 + MAX_STATIONS) DO
    IF g_stations[stn_num].tank_id = 0 THEN
      stn_num := stn_num + 1;
      CONTINUE;
    END_IF;

    stn_x := g_stations[stn_num].x_position;
    IF stn_x > max_x THEN
      EXIT;
    END_IF;

    avoid_st := g_avoid_status[stn_num];

    IF avoid_st = AVOID_PASS THEN
      is_target := (stn_num = g_transporter[i].lift_station)
               OR  (stn_num = g_transporter[i].sink_station);
      IF is_target THEN
        IF current_x < stn_x THEN
          new_val := stn_x - avoid_dist;
          IF new_val < max_x THEN max_x := new_val; END_IF;
          right_s2_x := stn_x;
          has_right_s2 := TRUE;
        ELSE
          new_val := stn_x + avoid_dist;
          IF new_val > min_x THEN min_x := new_val; END_IF;
          left_s2_x := stn_x;
          has_left_s2 := TRUE;
        END_IF;
        EXIT;
      END_IF;
    END_IF;

    IF avoid_st = AVOID_BLOCK THEN
      IF current_x < stn_x THEN
        new_val := stn_x - avoid_dist;
        IF new_val < max_x THEN max_x := new_val; END_IF;
        right_s2_x := stn_x;
        has_right_s2 := TRUE;
      ELSE
        new_val := stn_x + avoid_dist;
        IF new_val > min_x THEN min_x := new_val; END_IF;
        left_s2_x := stn_x;
        has_left_s2 := TRUE;
      END_IF;
      EXIT;
    END_IF;

    stn_num := stn_num + 1;
  END_WHILE;

  (* Conflict resolution: trapped between two BLOCK stations *)
  IF (min_x >= max_x) AND has_left_s2 AND has_right_s2 THEN
    midpoint := (left_s2_x + right_s2_x) / 2.0;
    min_x := midpoint - 5.0;
    max_x := midpoint + 5.0;
  END_IF;

  g_transporter[i].x_min_limit := min_x;
  g_transporter[i].x_max_limit := max_x;
END_FOR;

(* ================================================================
   STEP 2.0: Basic safety distance — current positions
   Every active transporter pushes neighbors away by x_avoid_mm.
   ================================================================ *)
FOR i := 1 TO TRANSPORTERS DO
  IF NOT g_transporter[i].active THEN
    CONTINUE;
  END_IF;

  current_x := INT_TO_REAL(REAL_TO_INT(g_transporter[i].x_mm + 0.5));
  current_y := g_transporter[i].y_mm;
  avoid_dist := g_cfg[i].x_avoid_mm;

  FOR j := 1 TO TRANSPORTERS DO
    IF j = i THEN CONTINUE; END_IF;
    IF NOT g_transporter[j].active THEN CONTINUE; END_IF;

    (* Skip transporters on different line (y-position check, matches JS Step 2.0) *)
    other_y := g_transporter[j].y_mm;
    IF ABS(other_y - current_y) >= 1.0 THEN CONTINUE; END_IF;

    other_x := INT_TO_REAL(REAL_TO_INT(g_transporter[j].x_mm + 0.5));

    IF other_x > current_x THEN
      (* j is to the RIGHT of i — restrict j's x_min *)
      new_val := current_x + avoid_dist;
      IF new_val > g_transporter[j].x_min_limit THEN
        g_transporter[j].x_min_limit := new_val;
      END_IF;
    ELSIF other_x < current_x THEN
      (* j is to the LEFT of i — restrict j's x_max *)
      new_val := current_x - avoid_dist;
      IF new_val < g_transporter[j].x_max_limit THEN
        g_transporter[j].x_max_limit := new_val;
      END_IF;
    END_IF;
  END_FOR;
END_FOR;

(* ================================================================
   STEP 2.2: Priority-based collision avoidance
   ================================================================ *)

(* --- 2.2.1: Build sorted array of active transporters by x-position --- *)
n_active := 0;
FOR i := 1 TO TRANSPORTERS DO
  IF g_transporter[i].active THEN
    n_active := n_active + 1;
    w_idx[n_active] := i;
    w_xpos[n_active] := INT_TO_REAL(REAL_TO_INT(g_transporter[i].x_mm + 0.5));
    w_phase[n_active] := g_transporter[i].phase;
    w_status[n_active] := g_transporter[i].status;
    w_ypos[n_active] := g_transporter[i].y_mm;
    w_target[n_active] := g_transporter[i].final_target_x;
    w_avoid[n_active] := g_cfg[i].x_avoid_mm;
  END_IF;
END_FOR;

(* Selection sort by x-position (ascending) *)
FOR i := 1 TO n_active - 1 DO
  min_idx := i;
  FOR j := i + 1 TO n_active DO
    IF w_xpos[j] < w_xpos[min_idx] THEN
      min_idx := j;
    END_IF;
  END_FOR;
  IF min_idx <> i THEN
    tmp_int := w_idx[i];    w_idx[i] := w_idx[min_idx];    w_idx[min_idx] := tmp_int;
    tmp_real := w_xpos[i];  w_xpos[i] := w_xpos[min_idx];  w_xpos[min_idx] := tmp_real;
    tmp_int := w_phase[i];  w_phase[i] := w_phase[min_idx]; w_phase[min_idx] := tmp_int;
    tmp_int := w_status[i]; w_status[i] := w_status[min_idx]; w_status[min_idx] := tmp_int;
    tmp_real := w_ypos[i];  w_ypos[i] := w_ypos[min_idx];  w_ypos[min_idx] := tmp_real;
    tmp_real := w_target[i]; w_target[i] := w_target[min_idx]; w_target[min_idx] := tmp_real;
    tmp_real := w_avoid[i];  w_avoid[i] := w_avoid[min_idx];  w_avoid[min_idx] := tmp_real;
  END_IF;
END_FOR;

(* --- 2.2.2: Calculate canEvade and priority --- *)
FOR i := 1 TO n_active DO
  k := w_idx[i];

  (* canEvade rules (from JS specification):
     RULE 1: status < 3 → not in automatic mode, cannot evade
     RULE 2: status = 4 AND phase ∈ {2,4} → Z-movement, cannot evade
     RULE 3: working area too small → cannot evade *)
  w_can_evade[i] := TRUE;
  IF w_status[i] < 3 THEN
    w_can_evade[i] := FALSE;
  END_IF;
  IF (w_status[i] = 4) AND ((w_phase[i] = 2) OR (w_phase[i] = 4)) THEN
    w_can_evade[i] := FALSE;
  END_IF;
  work_area := g_transporter[k].x_max_limit - g_transporter[k].x_min_limit;
  IF work_area < MIN_WORK_AREA THEN
    w_can_evade[i] := FALSE;
  END_IF;

  w_priority[i] := TWA_CalcPriority(
    i_phase := w_phase[i],
    i_can_evade := w_can_evade[i],
    i_x_pos := w_xpos[i],
    i_x_target := w_target[i]
  );
END_FOR;

(* Skip Steps 2.2.3-2.2.5 if fewer than 2 active transporters *)
IF n_active >= 2 THEN

  (* --- 2.2.3: Priority restrictions (higher priority → lower priority) --- *)
  FOR i := 1 TO n_active DO
    (* Skip idle transporters — they don't set priority restrictions *)
    IF w_phase[i] = 0 THEN CONTINUE; END_IF;

    FOR j := 1 TO n_active DO
      IF i = j THEN CONTINUE; END_IF;
      (* Skip transporters on different line *)
      IF ABS(w_ypos[i] - w_ypos[j]) >= 1.0 THEN CONTINUE; END_IF;

      (* Determine if i has higher priority than j *)
      a_wins := FALSE;
      IF w_priority[i] > w_priority[j] THEN
        a_wins := TRUE;
      ELSIF (w_priority[i] = w_priority[j]) AND (w_idx[i] < w_idx[j]) THEN
        a_wins := TRUE;
      END_IF;

      IF NOT a_wins THEN CONTINUE; END_IF;

      (* Higher priority transporter uses target for phase 1/3, else current pos *)
      IF (w_phase[i] = 1) OR (w_phase[i] = 3) THEN
        restrict_x := w_target[i];
      ELSE
        restrict_x := w_xpos[i];
      END_IF;

      k := w_idx[j];
      cur_min := g_transporter[k].x_min_limit;
      cur_max := g_transporter[k].x_max_limit;

      IF w_xpos[i] < w_xpos[j] THEN
        (* i is LEFT, j is RIGHT — i sets j's x_min *)
        (* Count same-line transporters between i and j *)
        between := 0;
        FOR stn_num := i + 1 TO j - 1 DO
          IF ABS(w_ypos[stn_num] - w_ypos[i]) < 1.0 THEN between := between + 1; END_IF;
        END_FOR;
        chain_ofs := w_avoid[i] + INT_TO_REAL(between) * (MIN_WORK_AREA + w_avoid[i]);
        new_val := restrict_x + chain_ofs;

        IF new_val > cur_min THEN
          IF new_val <= (cur_max - MIN_WORK_AREA) THEN
            g_transporter[k].x_min_limit := new_val;
          ELSE
            adjusted := cur_max - MIN_WORK_AREA;
            IF adjusted > cur_min THEN
              g_transporter[k].x_min_limit := adjusted;
            END_IF;
          END_IF;
        END_IF;

      ELSIF w_xpos[i] > w_xpos[j] THEN
        (* i is RIGHT, j is LEFT — i sets j's x_max *)
        (* Count same-line transporters between j and i *)
        between := 0;
        FOR stn_num := j + 1 TO i - 1 DO
          IF ABS(w_ypos[stn_num] - w_ypos[i]) < 1.0 THEN between := between + 1; END_IF;
        END_FOR;
        chain_ofs := w_avoid[i] + INT_TO_REAL(between) * (MIN_WORK_AREA + w_avoid[i]);
        new_val := restrict_x - chain_ofs;

        IF new_val < cur_max THEN
          IF new_val >= (cur_min + MIN_WORK_AREA) THEN
            g_transporter[k].x_max_limit := new_val;
          ELSE
            adjusted := cur_min + MIN_WORK_AREA;
            IF adjusted < cur_max THEN
              g_transporter[k].x_max_limit := adjusted;
            END_IF;
          END_IF;
        END_IF;
      END_IF;
    END_FOR;
  END_FOR;

  (* --- 2.2.4: Bidirectional safety (both moving same direction) --- *)
  FOR i := 1 TO n_active - 1 DO
    j := i + 1;
    (* i = left (smaller x), j = right (larger x) — sorted array *)

    (* Skip if not on same line *)
    IF ABS(w_ypos[i] - w_ypos[j]) >= 1.0 THEN CONTINUE; END_IF;

    left_right := ((w_phase[i] = 1) OR (w_phase[i] = 3)) AND (w_target[i] > w_xpos[i]);
    right_right := ((w_phase[j] = 1) OR (w_phase[j] = 3)) AND (w_target[j] > w_xpos[j]);
    left_left := ((w_phase[i] = 1) OR (w_phase[i] = 3)) AND (w_target[i] < w_xpos[i]);
    right_left := ((w_phase[j] = 1) OR (w_phase[j] = 3)) AND (w_target[j] < w_xpos[j]);

    IF left_right AND right_right THEN
      (* Both moving right — left chasing right *)
      safety_val := w_xpos[i] + w_avoid[i];
      k := w_idx[j];
      IF safety_val > g_transporter[k].x_min_limit THEN
        g_transporter[k].x_min_limit := safety_val;
      END_IF;
    END_IF;

    IF left_left AND right_left THEN
      (* Both moving left — right chasing left *)
      safety_val := w_xpos[j] - w_avoid[j];
      k := w_idx[i];
      IF safety_val < g_transporter[k].x_max_limit THEN
        g_transporter[k].x_max_limit := safety_val;
      END_IF;
    END_IF;
  END_FOR;

  (* --- 2.2.5: Validate limits (trap detection) --- *)
  FOR i := 1 TO n_active DO
    k := w_idx[i];
    IF g_transporter[k].x_min_limit > g_transporter[k].x_max_limit THEN
      (* Trapped — lock in place *)
      g_transporter[k].x_min_limit := g_transporter[k].x_mm;
      g_transporter[k].x_max_limit := g_transporter[k].x_mm;
    END_IF;
  END_FOR;

END_IF;  (* n_active >= 2 *)

END_FUNCTION_BLOCK

(* ---- config.st ---- *)
(* ============================================================
   config.st — PLC Configuration / Resource / Task
   ============================================================ *)

CONFIGURATION Config0
  RESOURCE Res0 ON PLC
    TASK task0(INTERVAL := T#20ms, PRIORITY := 0);
    PROGRAM instance0 WITH task0 : PLC_PRG;
  END_RESOURCE
END_CONFIGURATION

(* ---- plc_prg.st ---- *)
(* ============================================================
   plc_prg.st — Main program: config upload + transport cycle
   ============================================================ *)

PROGRAM PLC_PRG
VAR_EXTERNAL CONSTANT
    TRANSPORTERS : INT;
END_VAR

VAR_EXTERNAL
  g_station_count    : INT;
  g_stations         : ARRAY[101..125] OF STATION_T;
  g_cfg              : ARRAY[1..TRANSPORTERS] OF TRANSPORTER_CFG_T;
  g_transporter      : ARRAY[1..TRANSPORTERS] OF STC_TRANSPORTER_T;
  (* Modbus output: transporter 1 *)
  qw_t1_x_mm    : INT;
  qw_t1_z_mm    : INT;
  qw_t1_vel_x10 : INT;
  qw_t1_phase   : INT;
  qw_t1_z_stage : INT;
  qw_t1_cur_st  : INT;
  qw_t1_lift_tgt : INT;
  qw_t1_sink_tgt : INT;
  qw_t1_active  : INT;
  (* Modbus output: transporter 2 *)
  qw_t2_x_mm    : INT;
  qw_t2_z_mm    : INT;
  qw_t2_vel_x10 : INT;
  qw_t2_phase   : INT;
  qw_t2_z_stage : INT;
  qw_t2_cur_st  : INT;
  qw_t2_lift_tgt : INT;
  qw_t2_sink_tgt : INT;
  qw_t2_active  : INT;
  (* Modbus output: status *)
  qw_station_cnt : INT;
  qw_init_done   : INT;
  qw_cycle_cnt   : INT;
  (* Modbus input: move commands *)
  iw_cmd_start_1 : INT;
  iw_cmd_lift_1  : INT;
  iw_cmd_sink_1  : INT;
  iw_cmd_start_2 : INT;
  iw_cmd_lift_2  : INT;
  iw_cmd_sink_2  : INT;
  (* Config upload protocol *)
  iw_cfg_seq     : INT;
  iw_cfg_cmd     : INT;
  iw_cfg_param   : INT;
  iw_cfg_d0      : INT;
  iw_cfg_d1      : INT;
  iw_cfg_d2      : INT;
  iw_cfg_d3      : INT;
  iw_cfg_d4      : INT;
  iw_cfg_d5      : INT;
  iw_cfg_d6      : INT;
  qw_cfg_ack     : INT;
  (* Units array *)
  g_units        : ARRAY[1..10] OF UNIT_T;
  (* Modbus output: units QW22..QW61 *)
  qw_u1_loc  : INT;
  qw_u1_status  : INT;
  qw_u1_state  : INT;
  qw_u1_target  : INT;
  qw_u2_loc  : INT;
  qw_u2_status  : INT;
  qw_u2_state  : INT;
  qw_u2_target  : INT;
  qw_u3_loc  : INT;
  qw_u3_status  : INT;
  qw_u3_state  : INT;
  qw_u3_target  : INT;
  qw_u4_loc  : INT;
  qw_u4_status  : INT;
  qw_u4_state  : INT;
  qw_u4_target  : INT;
  qw_u5_loc  : INT;
  qw_u5_status  : INT;
  qw_u5_state  : INT;
  qw_u5_target  : INT;
  qw_u6_loc  : INT;
  qw_u6_status  : INT;
  qw_u6_state  : INT;
  qw_u6_target  : INT;
  qw_u7_loc  : INT;
  qw_u7_status  : INT;
  qw_u7_state  : INT;
  qw_u7_target  : INT;
  qw_u8_loc  : INT;
  qw_u8_status  : INT;
  qw_u8_state  : INT;
  qw_u8_target  : INT;
  qw_u9_loc  : INT;
  qw_u9_status  : INT;
  qw_u9_state  : INT;
  qw_u9_target  : INT;
  qw_u10_loc : INT;
  qw_u10_status : INT;
  qw_u10_state : INT;
  qw_u10_target : INT;
  qw_unit_ack  : INT;
  (* Modbus output: batch data QW65..QW104 *)
  qw_b1_code  : INT;  qw_b1_state  : INT;  qw_b1_prog  : INT;  qw_b1_stage  : INT;
  qw_b2_code  : INT;  qw_b2_state  : INT;  qw_b2_prog  : INT;  qw_b2_stage  : INT;
  qw_b3_code  : INT;  qw_b3_state  : INT;  qw_b3_prog  : INT;  qw_b3_stage  : INT;
  qw_b4_code  : INT;  qw_b4_state  : INT;  qw_b4_prog  : INT;  qw_b4_stage  : INT;
  qw_b5_code  : INT;  qw_b5_state  : INT;  qw_b5_prog  : INT;  qw_b5_stage  : INT;
  qw_b6_code  : INT;  qw_b6_state  : INT;  qw_b6_prog  : INT;  qw_b6_stage  : INT;
  qw_b7_code  : INT;  qw_b7_state  : INT;  qw_b7_prog  : INT;  qw_b7_stage  : INT;
  qw_b8_code  : INT;  qw_b8_state  : INT;  qw_b8_prog  : INT;  qw_b8_stage  : INT;
  qw_b9_code  : INT;  qw_b9_state  : INT;  qw_b9_prog  : INT;  qw_b9_stage  : INT;
  qw_b10_code : INT;  qw_b10_state : INT;  qw_b10_prog : INT;  qw_b10_stage : INT;
  (* Modbus input: unit write command *)
  iw_unit_seq    : INT;
  iw_unit_id     : INT;
  iw_unit_loc    : INT;
  iw_unit_status : INT;
  iw_unit_state  : INT;
  iw_unit_target : INT;
  (* Batch and program arrays *)
  g_batches      : ARRAY[1..10] OF BATCH_T;
  g_programs     : ARRAY[1..10] OF TREATMENT_PROGRAM_T;
  g_avoid_status : ARRAY[101..125] OF INT;
  (* Modbus input: batch write protocol *)
  iw_batch_seq     : INT;
  iw_batch_unit    : INT;
  iw_batch_code    : INT;
  iw_batch_state   : INT;
  iw_batch_prog_id : INT;
  qw_batch_ack     : INT;
  (* Modbus input: program stage write protocol *)
  iw_prog_seq      : INT;
  iw_prog_unit     : INT;
  iw_prog_stage    : INT;
  iw_prog_s1       : INT;
  iw_prog_s2       : INT;
  iw_prog_s3       : INT;
  iw_prog_s4       : INT;
  iw_prog_s5       : INT;
  iw_prog_min_time : INT;
  iw_prog_max_time : INT;
  iw_prog_cal_time : INT;
  qw_prog_ack      : INT;
  (* Unix time *)
  g_time_s    : LINT;
  iw_time_hi  : INT;
  iw_time_lo  : INT;
  (* Task scheduler globals *)
  g_schedule  : ARRAY[1..10] OF TSK_SCHEDULE_T;
  g_tasks     : ARRAY[1..TRANSPORTERS] OF TSK_QUEUE_T;
  (* Calibration *)
  g_cal       : ARRAY[1..TRANSPORTERS] OF CALIBRATION_T;
  g_cal_active : BOOL;
  (* Calibration output registers *)
  qw_cal_step     : INT;
  qw_cal_tid      : INT;
  qw_cal_t1_lift_wet : INT;
  qw_cal_t1_sink_wet : INT;
  qw_cal_t1_lift_dry : INT;
  qw_cal_t1_sink_dry : INT;
  qw_cal_t1_x_acc    : INT;
  qw_cal_t1_x_dec    : INT;
  qw_cal_t1_x_max    : INT;
  qw_cal_t2_lift_wet : INT;
  qw_cal_t2_sink_wet : INT;
  qw_cal_t2_lift_dry : INT;
  qw_cal_t2_sink_dry : INT;
  qw_cal_t2_x_acc    : INT;
  qw_cal_t2_x_dec    : INT;
  qw_cal_t2_x_max    : INT;
  qw_cal_t3_lift_wet : INT;
  qw_cal_t3_sink_wet : INT;
  qw_cal_t3_lift_dry : INT;
  qw_cal_t3_sink_dry : INT;
  qw_cal_t3_x_acc    : INT;
  qw_cal_t3_x_dec    : INT;
  qw_cal_t3_x_max    : INT;
END_VAR
VAR
  init_done      : BOOL := FALSE;
  last_cfg_seq   : INT := 0;
  last_unit_seq  : INT := 0;
  last_batch_seq : INT := 0;
  last_prog_seq  : INT := 0;
  j              : INT;
  k              : INT;
  i              : INT;
  stn_num        : INT;
  idx          : INT;
  twa_calc     : TWA_FB_CalcLimits;
  lookup       : STC_FB_FindStation;
  clear_cfg    : SIM_FB_ClearConfig;
  cycle_count  : INT;
  main_sched   : STC_FB_MainScheduler;
  run_tasks    : SIM_FB_RunTasks;
  calibrate    : STC_FB_Calibrate;
  cal_cmd      : INT := 0;
  (* Time-keeping vars *)
  time_hi        : LINT;
  time_lo        : LINT;
  time_cycle_cnt : INT := 0;      (* counts 20ms cycles, resets at 50 = 1 s *)
  last_sync_hi   : INT := 0;      (* previous gateway iw_time_hi — for change detect *)
  last_sync_lo   : INT := 0;      (* previous gateway iw_time_lo *)
END_VAR
(* ============================================================
   CONFIG UPLOAD HANDLER
   Gateway writes station data one at a time via Modbus IW regs.
   Sequence number change triggers processing.
   cmd=1: write_station  cmd=2: init  cmd=3: clear_all
   ============================================================ *)
IF iw_cfg_seq <> last_cfg_seq THEN
  last_cfg_seq := iw_cfg_seq;

  IF iw_cfg_cmd = 3 THEN
    (* --- Clear all config data --- *)
    clear_cfg();
    init_done := FALSE;
    qw_init_done := 0;
    qw_station_cnt := 0;
    qw_cfg_ack := iw_cfg_seq;

  ELSIF iw_cfg_cmd = 1 THEN
    (* --- Write one station to g_stations array --- *)
    IF (iw_cfg_param >= 101) AND (iw_cfg_param <= 125) THEN
      g_stations[iw_cfg_param].tank_id       := iw_cfg_d0;
      g_stations[iw_cfg_param].x_position    := INT_TO_REAL(iw_cfg_d1);
      g_stations[iw_cfg_param].y_position    := INT_TO_REAL(iw_cfg_d2);
      g_stations[iw_cfg_param].z_position    := INT_TO_REAL(iw_cfg_d3);
      g_stations[iw_cfg_param].stn_function  := iw_cfg_d4;
      IF (iw_cfg_d4 = 1) OR (iw_cfg_d4 = 11) THEN
        g_stations[iw_cfg_param].stn_type := 1;   (* wet *)
      ELSE
        g_stations[iw_cfg_param].stn_type := 0;   (* dry *)
      END_IF;
      g_stations[iw_cfg_param].dropping_time := INT_TO_REAL(iw_cfg_d5) / 10.0;
      g_stations[iw_cfg_param].device_delay  := INT_TO_REAL(iw_cfg_d6) / 10.0;
    END_IF;
    qw_cfg_ack := iw_cfg_seq;

  ELSIF iw_cfg_cmd = 4 THEN
    (* --- Write transporter physics page 1 --- *)
    (* param = transporter_id (1..3)
       d0 = x_min_limit mm      d1 = x_max_limit mm
       d2 = x_accel_s × 10      d3 = x_decel_s × 10
       d4 = x_max_mm_s           d5 = z_total_mm
       d6 = avoid_mm *)
    j := iw_cfg_param;
    IF (j >= 1) AND (j <= 3) THEN
      g_cfg[j].x_min_limit          := INT_TO_REAL(iw_cfg_d0);
      g_cfg[j].x_max_limit          := INT_TO_REAL(iw_cfg_d1);
      g_cfg[j].phys2d.x_accel_s     := INT_TO_REAL(iw_cfg_d2) / 10.0;
      g_cfg[j].phys2d.x_decel_s     := INT_TO_REAL(iw_cfg_d3) / 10.0;
      g_cfg[j].phys2d.x_max_mm_s    := INT_TO_REAL(iw_cfg_d4);
      g_cfg[j].phys2d.z_total_mm    := INT_TO_REAL(iw_cfg_d5);
      g_cfg[j].phys2d.avoid_mm      := INT_TO_REAL(iw_cfg_d6);
      g_cfg[j].x_avoid_mm           := INT_TO_REAL(iw_cfg_d6);
    END_IF;
    qw_cfg_ack := iw_cfg_seq;

  ELSIF iw_cfg_cmd = 5 THEN
    (* --- Write transporter physics page 2 --- *)
    (* param = transporter_id (1..3)
       d0 = z_slow_dry_mm        d1 = z_slow_wet_mm
       d2 = z_slow_end_mm        d3 = z_slow_mm_s
       d4 = z_fast_mm_s          d5 = drip_delay_s × 10
       d6 = (reserved) *)
    j := iw_cfg_param;
    IF (j >= 1) AND (j <= 3) THEN
      g_cfg[j].phys2d.z_slow_dry_mm := INT_TO_REAL(iw_cfg_d0);
      g_cfg[j].phys2d.z_slow_wet_mm := INT_TO_REAL(iw_cfg_d1);
      g_cfg[j].phys2d.z_slow_end_mm := INT_TO_REAL(iw_cfg_d2);
      g_cfg[j].phys2d.z_slow_mm_s   := INT_TO_REAL(iw_cfg_d3);
      g_cfg[j].phys2d.z_fast_mm_s   := INT_TO_REAL(iw_cfg_d4);
      g_cfg[j].phys2d.drip_delay_s  := INT_TO_REAL(iw_cfg_d5) / 10.0;
    END_IF;
    qw_cfg_ack := iw_cfg_seq;

  ELSIF iw_cfg_cmd = 6 THEN
    (* --- Write transporter task area --- *)
    (* param = transporter_id × 10 + area_index
       e.g. 11 = transporter 1 area 1, 23 = transporter 2 area 3
       d0 = min_lift   d1 = max_lift
       d2 = min_sink   d3 = max_sink *)
    j := iw_cfg_param / 10;
    k := iw_cfg_param MOD 10;
    IF (j >= 1) AND (j <= 3) AND (k >= 1) AND (k <= 4) THEN
      g_cfg[j].task_area[k].min_lift := iw_cfg_d0;
      g_cfg[j].task_area[k].max_lift := iw_cfg_d1;
      g_cfg[j].task_area[k].min_sink := iw_cfg_d2;
      g_cfg[j].task_area[k].max_sink := iw_cfg_d3;
    END_IF;
    qw_cfg_ack := iw_cfg_seq;

  ELSIF iw_cfg_cmd = 7 THEN
    (* --- Calibration plan for one transporter --- *)
    (* param = transporter_id (1..3)
       d0 = wet_station   d1 = dry_station *)
    j := iw_cfg_param;
    IF (j >= 1) AND (j <= 3) THEN
      g_cal[j].wet_station := iw_cfg_d0;
      g_cal[j].dry_station := iw_cfg_d1;
    END_IF;
    qw_cfg_ack := iw_cfg_seq;

  ELSIF iw_cfg_cmd = 8 THEN
    (* --- Calibration control --- *)
    (* param: 1=start, 2=calculate, 3=abort *)
    cal_cmd := iw_cfg_param;
    qw_cfg_ack := iw_cfg_seq;

  ELSIF iw_cfg_cmd = 2 THEN
    (* --- Finish init: all config uploaded, init transporter states --- *)
    g_station_count := iw_cfg_param;

    FOR i := 1 TO TRANSPORTERS DO
      (* Active if task_area[1] has non-zero stations *)
      IF g_cfg[i].task_area[1].min_lift > 0 THEN
        g_transporter[i].active := TRUE;
      ELSE
        g_transporter[i].active := FALSE;
      END_IF;
      g_transporter[i].phase := 0;
      g_transporter[i].z_stage := 0;
      g_transporter[i].vel_x := 0.0;
      g_transporter[i].z_timer_s := 0.0;
      g_transporter[i].x_min_limit := g_cfg[i].x_min_limit;
      g_transporter[i].x_max_limit := g_cfg[i].x_max_limit;

      (* Start position: use task_area[1].min_lift as start station *)
      IF g_cfg[i].task_area[1].min_lift > 0 THEN
        stn_num := g_cfg[i].task_area[1].min_lift;
      ELSE
        stn_num := 0;
      END_IF;
      lookup(station_number := stn_num);
      IF lookup.found THEN
        g_transporter[i].x_mm := lookup.x_mm;
        g_transporter[i].current_station := stn_num;
      ELSE
        g_transporter[i].x_mm := 0.0;
        g_transporter[i].current_station := 0;
      END_IF;
      g_transporter[i].z_mm := 0.0;
    END_FOR;

    init_done := TRUE;
    qw_cfg_ack := iw_cfg_seq;
  END_IF;
END_IF;

(* ============================================================
   MAIN TRANSPORT CYCLE — only runs when init_done
   ============================================================ *)
IF init_done THEN

(* Calculate transporter working areas (X-limits) every cycle *)
twa_calc();

(* ── Unix time maintenance ── *)
(* PLC keeps g_time_s by incrementing +1 every 50 cycles (50 × 20 ms = 1 s).
   Gateway periodically writes reference unix seconds to QW160/QW161.
   When PLC detects the register values changed → sync to gateway time. *)
IF iw_time_hi <> last_sync_hi OR iw_time_lo <> last_sync_lo THEN
  (* Gateway wrote new reference time — sync *)
  time_hi := INT_TO_LINT(iw_time_hi);
  IF time_hi < LINT#0 THEN
    time_hi := time_hi + LINT#65536;
  END_IF;
  time_lo := INT_TO_LINT(iw_time_lo);
  IF time_lo < LINT#0 THEN
    time_lo := time_lo + LINT#65536;
  END_IF;
  g_time_s := time_hi * LINT#65536 + time_lo;
  last_sync_hi := iw_time_hi;
  last_sync_lo := iw_time_lo;
  time_cycle_cnt := 0;
ELSE
  (* Self-increment: +1 second every 50 cycles (50 × 20 ms) *)
  time_cycle_cnt := time_cycle_cnt + 1;
  IF time_cycle_cnt >= 50 THEN
    g_time_s := g_time_s + LINT#1;
    time_cycle_cnt := 0;
  END_IF;
END_IF;

(* ── Main Scheduler (TSK + DEP alternating cycles) ── *)
main_sched(i_run := init_done, i_time_s := g_time_s);

(* ── Execute transporter tasks (physics simulation) ── *)
run_tasks(i_run := init_done);

(* ── Calibration FB — issues test tasks, measures parameters ── *)
calibrate(i_run := init_done, i_cmd := cal_cmd);
cal_cmd := 0;   (* consumed after one cycle *)
g_cal_active := calibrate.o_active;

END_IF;  (* init_done *)

(* ============================================================
   UNIT WRITE HANDLER — gateway writes one unit at a time
   ============================================================ *)
IF iw_unit_seq <> last_unit_seq THEN
  last_unit_seq := iw_unit_seq;
  IF (iw_unit_id >= 1) AND (iw_unit_id <= 10) THEN
    g_units[iw_unit_id].location := iw_unit_loc;
    g_units[iw_unit_id].status   := iw_unit_status;
    g_units[iw_unit_id].state    := iw_unit_state;
    g_units[iw_unit_id].target   := iw_unit_target;
  END_IF;
  qw_unit_ack := iw_unit_seq;
END_IF;

(* ============================================================
   BATCH WRITE HANDLER — gateway writes batch data + program_id
   Also clears all stages of the treatment program for this unit.
   ============================================================ *)
IF iw_batch_seq <> last_batch_seq THEN
  last_batch_seq := iw_batch_seq;
  IF (iw_batch_unit >= 1) AND (iw_batch_unit <= 10) THEN
    g_batches[iw_batch_unit].batch_code := iw_batch_code;
    g_batches[iw_batch_unit].state      := iw_batch_state;
    g_batches[iw_batch_unit].prog_id    := iw_batch_prog_id;
    g_batches[iw_batch_unit].cur_stage      := 0;
    g_programs[iw_batch_unit].program_id := iw_batch_prog_id;
    (* Clear all stages *)
    FOR j := 1 TO 30 DO
      FOR k := 1 TO 5 DO
        g_programs[iw_batch_unit].stages[j].stations[k] := 0;
      END_FOR;
      g_programs[iw_batch_unit].stages[j].min_time := 0;
      g_programs[iw_batch_unit].stages[j].max_time := 0;
      g_programs[iw_batch_unit].stages[j].cal_time := 0;
    END_FOR;
  END_IF;
  qw_batch_ack := iw_batch_seq;
END_IF;

(* ============================================================
   PROGRAM STAGE WRITE HANDLER — gateway writes one stage at a time
   ============================================================ *)
IF iw_prog_seq <> last_prog_seq THEN
  last_prog_seq := iw_prog_seq;
  IF (iw_prog_unit >= 1) AND (iw_prog_unit <= 10) AND
     (iw_prog_stage >= 1) AND (iw_prog_stage <= 30) THEN
    g_programs[iw_prog_unit].stages[iw_prog_stage].stations[1] := iw_prog_s1;
    g_programs[iw_prog_unit].stages[iw_prog_stage].stations[2] := iw_prog_s2;
    g_programs[iw_prog_unit].stages[iw_prog_stage].stations[3] := iw_prog_s3;
    g_programs[iw_prog_unit].stages[iw_prog_stage].stations[4] := iw_prog_s4;
    g_programs[iw_prog_unit].stages[iw_prog_stage].stations[5] := iw_prog_s5;
    g_programs[iw_prog_unit].stages[iw_prog_stage].min_time := iw_prog_min_time;
    g_programs[iw_prog_unit].stages[iw_prog_stage].max_time := iw_prog_max_time;
    g_programs[iw_prog_unit].stages[iw_prog_stage].cal_time := iw_prog_cal_time;
  END_IF;
  qw_prog_ack := iw_prog_seq;
END_IF;

(* === MODBUS INPUT: Read commands → g_transporter command fields === *)
(* Note: task_id sync will be handled by SIM_FB_RunTasks later.
   For now, keep the old Modbus command interface working via direct write. *)
IF (iw_cmd_start_1 <> 0) AND (g_transporter[1].phase = 0) THEN
  g_transporter[1].task_id := g_time_s;
  g_transporter[1].lift_station := iw_cmd_lift_1;
  g_transporter[1].sink_station := iw_cmd_sink_1;
END_IF;
IF (iw_cmd_start_2 <> 0) AND (g_transporter[2].phase = 0) THEN
  g_transporter[2].task_id := g_time_s;
  g_transporter[2].lift_station := iw_cmd_lift_2;
  g_transporter[2].sink_station := iw_cmd_sink_2;
END_IF;

(* === MODBUS OUTPUT: Write transporter 1 state === *)
qw_t1_x_mm := REAL_TO_INT(g_transporter[1].x_mm);
qw_t1_z_mm := REAL_TO_INT(g_transporter[1].z_mm);
qw_t1_vel_x10 := REAL_TO_INT(g_transporter[1].vel_x * 10.0);
qw_t1_phase := g_transporter[1].phase;
qw_t1_z_stage := g_transporter[1].z_stage;
qw_t1_cur_st := g_transporter[1].current_station;
qw_t1_lift_tgt := g_transporter[1].lift_station;
qw_t1_sink_tgt := g_transporter[1].sink_station;
IF g_transporter[1].active THEN qw_t1_active := 1; ELSE qw_t1_active := 0; END_IF;

(* === MODBUS OUTPUT: Write transporter 2 state === *)
qw_t2_x_mm := REAL_TO_INT(g_transporter[2].x_mm);
qw_t2_z_mm := REAL_TO_INT(g_transporter[2].z_mm);
qw_t2_vel_x10 := REAL_TO_INT(g_transporter[2].vel_x * 10.0);
qw_t2_phase := g_transporter[2].phase;
qw_t2_z_stage := g_transporter[2].z_stage;
qw_t2_cur_st := g_transporter[2].current_station;
qw_t2_lift_tgt := g_transporter[2].lift_station;
qw_t2_sink_tgt := g_transporter[2].sink_station;
IF g_transporter[2].active THEN qw_t2_active := 1; ELSE qw_t2_active := 0; END_IF;

(* === MODBUS OUTPUT: Status registers === *)
qw_station_cnt := g_station_count;
IF init_done THEN qw_init_done := 1; ELSE qw_init_done := 0; END_IF;
cycle_count := cycle_count + 1;
IF cycle_count > 30000 THEN cycle_count := 0; END_IF;
qw_cycle_cnt := cycle_count;

(* Write unit data to Modbus output QW22..QW61 *)
qw_u1_loc    := g_units[1].location;
qw_u1_status := g_units[1].status;
qw_u1_state  := g_units[1].state;
qw_u1_target := g_units[1].target;
qw_u2_loc    := g_units[2].location;
qw_u2_status := g_units[2].status;
qw_u2_state  := g_units[2].state;
qw_u2_target := g_units[2].target;
qw_u3_loc    := g_units[3].location;
qw_u3_status := g_units[3].status;
qw_u3_state  := g_units[3].state;
qw_u3_target := g_units[3].target;
qw_u4_loc    := g_units[4].location;
qw_u4_status := g_units[4].status;
qw_u4_state  := g_units[4].state;
qw_u4_target := g_units[4].target;
qw_u5_loc    := g_units[5].location;
qw_u5_status := g_units[5].status;
qw_u5_state  := g_units[5].state;
qw_u5_target := g_units[5].target;
qw_u6_loc    := g_units[6].location;
qw_u6_status := g_units[6].status;
qw_u6_state  := g_units[6].state;
qw_u6_target := g_units[6].target;
qw_u7_loc    := g_units[7].location;
qw_u7_status := g_units[7].status;
qw_u7_state  := g_units[7].state;
qw_u7_target := g_units[7].target;
qw_u8_loc    := g_units[8].location;
qw_u8_status := g_units[8].status;
qw_u8_state  := g_units[8].state;
qw_u8_target := g_units[8].target;
qw_u9_loc    := g_units[9].location;
qw_u9_status := g_units[9].status;
qw_u9_state  := g_units[9].state;
qw_u9_target := g_units[9].target;
qw_u10_loc    := g_units[10].location;
qw_u10_status := g_units[10].status;
qw_u10_state  := g_units[10].state;
qw_u10_target := g_units[10].target;

(* Write batch data to Modbus output QW65..QW104 *)
qw_b1_code  := g_batches[1].batch_code;  qw_b1_state  := g_batches[1].state;  qw_b1_prog  := g_batches[1].prog_id;  qw_b1_stage  := g_batches[1].cur_stage;
qw_b2_code  := g_batches[2].batch_code;  qw_b2_state  := g_batches[2].state;  qw_b2_prog  := g_batches[2].prog_id;  qw_b2_stage  := g_batches[2].cur_stage;
qw_b3_code  := g_batches[3].batch_code;  qw_b3_state  := g_batches[3].state;  qw_b3_prog  := g_batches[3].prog_id;  qw_b3_stage  := g_batches[3].cur_stage;
qw_b4_code  := g_batches[4].batch_code;  qw_b4_state  := g_batches[4].state;  qw_b4_prog  := g_batches[4].prog_id;  qw_b4_stage  := g_batches[4].cur_stage;
qw_b5_code  := g_batches[5].batch_code;  qw_b5_state  := g_batches[5].state;  qw_b5_prog  := g_batches[5].prog_id;  qw_b5_stage  := g_batches[5].cur_stage;
qw_b6_code  := g_batches[6].batch_code;  qw_b6_state  := g_batches[6].state;  qw_b6_prog  := g_batches[6].prog_id;  qw_b6_stage  := g_batches[6].cur_stage;
qw_b7_code  := g_batches[7].batch_code;  qw_b7_state  := g_batches[7].state;  qw_b7_prog  := g_batches[7].prog_id;  qw_b7_stage  := g_batches[7].cur_stage;
qw_b8_code  := g_batches[8].batch_code;  qw_b8_state  := g_batches[8].state;  qw_b8_prog  := g_batches[8].prog_id;  qw_b8_stage  := g_batches[8].cur_stage;
qw_b9_code  := g_batches[9].batch_code;  qw_b9_state  := g_batches[9].state;  qw_b9_prog  := g_batches[9].prog_id;  qw_b9_stage  := g_batches[9].cur_stage;
qw_b10_code := g_batches[10].batch_code; qw_b10_state := g_batches[10].state; qw_b10_prog := g_batches[10].prog_id; qw_b10_stage := g_batches[10].cur_stage;

(* Write calibration status & results to Modbus QW170..QW192 *)
qw_cal_step := calibrate.o_step;
qw_cal_tid  := calibrate.o_tid;
(* T1 *)
qw_cal_t1_lift_wet := REAL_TO_INT(g_cal[1].lift_wet_s * 10.0);
qw_cal_t1_sink_wet := REAL_TO_INT(g_cal[1].sink_wet_s * 10.0);
qw_cal_t1_lift_dry := REAL_TO_INT(g_cal[1].lift_dry_s * 10.0);
qw_cal_t1_sink_dry := REAL_TO_INT(g_cal[1].sink_dry_s * 10.0);
qw_cal_t1_x_acc    := REAL_TO_INT(g_cal[1].x_accel_s * 10.0);
qw_cal_t1_x_dec    := REAL_TO_INT(g_cal[1].x_decel_s * 10.0);
qw_cal_t1_x_max    := REAL_TO_INT(g_cal[1].x_max_mm_s);
(* T2 *)
qw_cal_t2_lift_wet := REAL_TO_INT(g_cal[2].lift_wet_s * 10.0);
qw_cal_t2_sink_wet := REAL_TO_INT(g_cal[2].sink_wet_s * 10.0);
qw_cal_t2_lift_dry := REAL_TO_INT(g_cal[2].lift_dry_s * 10.0);
qw_cal_t2_sink_dry := REAL_TO_INT(g_cal[2].sink_dry_s * 10.0);
qw_cal_t2_x_acc    := REAL_TO_INT(g_cal[2].x_accel_s * 10.0);
qw_cal_t2_x_dec    := REAL_TO_INT(g_cal[2].x_decel_s * 10.0);
qw_cal_t2_x_max    := REAL_TO_INT(g_cal[2].x_max_mm_s);
(* T3 *)
qw_cal_t3_lift_wet := REAL_TO_INT(g_cal[3].lift_wet_s * 10.0);
qw_cal_t3_sink_wet := REAL_TO_INT(g_cal[3].sink_wet_s * 10.0);
qw_cal_t3_lift_dry := REAL_TO_INT(g_cal[3].lift_dry_s * 10.0);
qw_cal_t3_sink_dry := REAL_TO_INT(g_cal[3].sink_dry_s * 10.0);
qw_cal_t3_x_acc    := REAL_TO_INT(g_cal[3].x_accel_s * 10.0);
qw_cal_t3_x_dec    := REAL_TO_INT(g_cal[3].x_decel_s * 10.0);
qw_cal_t3_x_max    := REAL_TO_INT(g_cal[3].x_max_mm_s);
END_PROGRAM
